RoboDK station: project.rdk

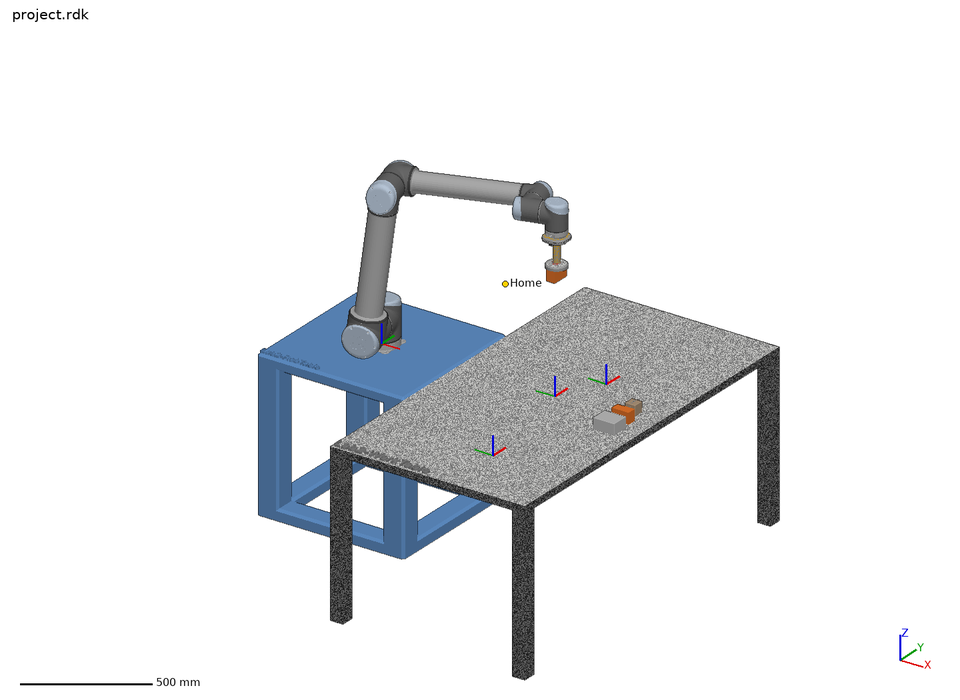
[picture v0: the station drawn from its stored meshes, robots at their saved joint values, targets as dots, program paths as lines]
Station project. Poses are relative to the parent item; angles as X-Y-Z fixed-axis rotations.
  - frame robot base at (200, 1000, 100) mm
    - robot robot: 6 axes, payload 10 kg, reach 1300 mm, repeatability 0.1 mm, weight 28.9 kg
        modified DH rows (alpha deg, a mm, theta deg, d mm): 0, 0, 0, 118; 90, 0, 180, 0; 0, 612.7, 0, 0; 0, 571.6, 0, 163.9; -90, 0, 0, 115.7; 90, 0, 180, 92.2
        joint limits [-360, -360, -360, -360, -360, -360] to [360, 360, 360, 360, 360, 360]; home [0, -90, -90, 0, 90, 0]; saved at [15.049, -97.194, -80.668, -92.138, 90, 105.049]
      - tool robotTool, TCP at (0, 0, 130) mm, size 100 x 100 x 133.5 mm, geometry from CostumTool.iges
        - object Box1 at (-20, -40, 0) mm, size 40 x 80 x 50 mm, geometry from Exquisite Snaget (1).stl
    - object RobTable at (0, 0, 0) mm, size 680 x 680 x 690 mm, geometry from RobTable.iges
    - target Home (Cartesian target) at (687.3, -163.9, 508.5) mm, rotated rx 180 ry 0 rz -90 deg; joints [0, -90, -90, -90, 90, 0] of robot
    - frame pickFrame at (800, 0, 0) mm, rotated rx 0 ry 0 rz 90 deg
      - frame placeFrameLeft at (-550, -100, 0) mm
      - frame placeFrameRight at (200, -100, 0) mm
      - object WoodBox at (30, -350, 0) mm, size 50 x 48 x 50 mm, geometry from WoodBox.iges
      - object Box1 at (-40, -370, 0) mm, size 40 x 80 x 50 mm, geometry from Exquisite Snaget (1).stl
      - object Box2 at (-150, -380, 0) mm, size 80 x 100 x 50 mm, geometry from Box.stl
    - object WorkTable at (800, 0, 0) mm, size 900 x 1680 x 742 mm, geometry from WorkTable.iges
